(* PLC project product_creator, Dassault Systèmes ControlBuild 2024x *)
(* stored: creationDateTime 2023-10-03T11:12:53-01:00 *)

(* This module simulates the creation of products. The creation can be : - pulsed - automatic and cyclic *)
FUNCTION_BLOCK equipment_library.product_creator
  VAR
    status_act_prod : DINT := 0;
    m11 : REAL := 1.0;
    m12 : REAL := 0.0;
    m13 : REAL := 0.0;
    m14 : REAL := 0.0;
    m21 : REAL := 0.0;
    m22 : REAL := 1.0;
    m23 : REAL := 0.0;
    m24 : REAL := 0.0;
    m31 : REAL := 0.0;
    m32 : REAL := 0.0;
    m33 : REAL := 1.0;
    m34 : REAL := 0.0;
    m41 : REAL := 0.0;
    m42 : REAL := 0.0;
    m43 : REAL := 0.0;
    m44 : REAL := 1.0;
    pbCreation : BOOL := false;
    productPresence : BOOL := false;
    idProd : DINT := 0;
    cntProd : DINT := 0;
    waitingTime : REAL := 10.0;
    oldIdProd : DINT := 0;
  END_VAR
  VAR CONSTANT
    gravitySpeed : REAL := 0.1;
    nbProdToCreate : INT := 1;
    pulsedMode : BOOL := true;
    pulseTime : REAL := 10.0;
    alignProductsToZ : BOOL := true;
    alignProductsToY : BOOL := false;
    alignProductsToX : BOOL := false;
  END_VAR


ACTION C_source_code:
/* ----------------------------------------------------------------	*/
/* Type : Model of Operative Behaviour					*/
/* Category :  Actors and Products						*/
/* Author : Dassault Systemes						*/
/* Update date : June 2018							*/
/* ----------------------------------------------------------------	*/
/* This module simulates the creation of products.			*/
/* The creation can be :							*/
/* - pulsed									*/
/* - automatic and cyclic							*/
/* ----------------------------------------------------------------	*/


int i;
 
if (!  pulsedMode) {
	waitingTime += CLOCK_PERIOD / 1000000.0;
	if (productPresence) waitingTime = 0.0;
}

/* ----------------------------------------------------------------	*/
/* Request for creation of a product at the same location that the	*/
/* creation module.								*/
/* To avoid inopportune stacking, the creation of a new product is	*/
/* forbidden when there is already one in the creation area.		*/
/* ----------------------------------------------------------------	*/

if ((pbCreation ||  ((waitingTime>= pulseTime) && ! pulsedMode)) && ! productPresence) {
	waitingTime = 0.0;
	for (i=0;i<nbProdToCreate;i++) {
		if (alignProductsToX) {
			idProd=prodNew(equipment_library__box, getPositionX(myself), getPositionY(myself), getPositionZ(myself), getSizeX(myself), getSizeY(myself), getSizeZ(myself));
			if (idProd >= 0)
				rotateTo(idProd, getAngleX(myself), getAngleY(myself), getAngleZ(myself), getPositionX(idProd), getPositionY(idProd),getPositionZ(idProd));
			if (i>0) moveRelativeAnotherXBy(idProd, oldIdProd , (getSizeX(myself)*i));

			oldIdProd = idProd;
		}
		if (alignProductsToY) {
			idProd=prodNew(equipment_library__box, getPositionX(myself), getPositionY(myself), getPositionZ(myself), getSizeX(myself), getSizeY(myself), getSizeZ(myself));
			if (idProd >= 0)
				rotateTo(idProd, getAngleX(myself), getAngleY(myself), getAngleZ(myself), getPositionX(idProd), getPositionY(idProd),getPositionZ(idProd));
			if (i>0) moveRelativeAnotherYBy(idProd, oldIdProd , (getSizeY(myself)*i));
			oldIdProd = idProd;
		}
		if (alignProductsToZ) {
			idProd=prodNew(equipment_library__box, getPositionX(myself), getPositionY(myself), getPositionZ(myself)+(getSizeZ(myself)*i), getSizeX(myself), getSizeY(myself), getSizeZ(myself));
			if (idProd >= 0)
				rotateTo(idProd, getAngleX(myself), getAngleY(myself), getAngleZ(myself), getPositionX(idProd), getPositionY(idProd),getPositionZ(idProd));
		}
		
		if (idProd >= 0) {
			cntProd++;
			var(idProd, equipment_library__box__gravitySpeed)=gravitySpeed;
			var(idProd, equipment_library__box__number)=cntProd;
		}
	}
}


/* ----------------------------------------------------------------	*/
/* Reset information on product presence					*/
/* ----------------------------------------------------------------	*/
productPresence=0;

/* ----------------------------------------------------------------	*/
/* Reset of the manual request for creation				*/
/* ----------------------------------------------------------------	*/
pbCreation=0;
END_ACTION

ACTION C_header:
#include "equipment_library/functional/box/box.h"
END_ACTION
END_FUNCTION_BLOCK
